// TIA Portal V19 export
TYPE "BurkettType8691_UDTNest"
   STRUCT
      OP : "OP_Int";
      Commands : "IF_Commands";
      "IF" : "Burkett 8691 REV.3";
   END_STRUCT;
END_TYPE
